{attribute 'linkalways'} 
{attribute 'no_explicit_call' := 'This FB is a CLASS and must be accessed using methods or properties'}
{attribute 'enable_dynamic_creation'}
FUNCTION_BLOCK Node_F_VN_AppendToContainer_ITcVnImage EXTENDS VisionNode
VAR
    ipElement : _ITcVnImage;
    ipContainer : _ITcVnContainer;
    hrPrev : _HRESULT(S_OK);
	hresult : _HRESULT(S_OK);
END_VAR

METHOD PUBLIC  Clone : I_Node
VAR
	pNode : POINTER TO Node_F_VN_AppendToContainer_ITcVnImage;
END_VAR
pNode := __NEW(Node_F_VN_AppendToContainer_ITcVnImage);
Clone := pNode^;
END_METHOD

METHOD FB_init : BOOL
VAR_INPUT
	bInitRetains : BOOL; // if TRUE, the retain variables are initialized (warm start / cold start)
	bInCopyCode : BOOL;  // if TRUE, the instance afterwards gets moved into the copy code (online change)
END_VAR
AddInput('ipElement', ipElement);
AddInput('ipContainer', ipContainer);
AddInput('hrPrev', hrPrev);
AddOutput('ipContainer', ipContainer);
AddOutput('hresult',hresult);
END_METHOD

METHOD PROTECTED OnExecute
hresult.Value := F_VN_AppendToContainer_ITcVnImage(
    ipElement := ipElement.Value,
	ipContainer := ipContainer.Value,
	hrPrev:= hrPrev.Value);
END_METHOD

METHOD PUBLIC PreExecutionCheck
VAR_INPUT
	Check : I_PreExecutionChecks;
END_VAR
Check.IsTrue(ipContainer.IsValid, 'ipContainer must be a valid container');
Check.IsTrue(ipContainer.IsType(TC_GLOBAL_CONST_LIST.ContainerType_Vector_ITcVnImage), 'ipContainer contains incorrect type');
END_METHOD

END_FUNCTION_BLOCK

(* stored: Version 1.1.0.1, ProductVersion 3.1.4026.13
   POU Node_F_VN_AppendToContainer_ITcVnImage: Id {94499260-a594-4876-a97f-2e8b3f45c15c}, SpecialFunc None
   Folder Constructor: Id {e61c9d1d-f9ec-4051-b98d-28da625769bb}
   Method Clone: Id {7317c3cb-e62b-41e6-8454-e6fd937a53b1}
   Method FB_init: Id {b51808a5-eaab-4dce-9443-b13187a9375c}
   Method OnExecute: Id {cbd3d27a-4774-4b22-9239-7462adcb4730}
   Method PreExecutionCheck: Id {2fde3047-ac62-4f4a-9723-dfc8a6c2fc04} *)
